(* CoDeSys 2.3 export: VARST.EXP *)

(* Data type *)
TYPE VarST :
STRUCT
    pby:      POINTER TO BYTE;
    type_:    VarType;
END_STRUCT
END_TYPE
